// SIMATIC S7-200 project (STEP 7-Micro/WIN), CPU 222 REL 02.01

SYMBOL_TABLE USER1
E0               M0.0     // ESTADO 0
E1               M0.1     // ESTADO 1
E2               M0.2     // ESTADO 2
E3               M0.3     // ESTADO 3
E4               M0.4     // ESTADO 4
E5               M0.5     // ESTADO 5
E6               M0.6     // ESTADO 6
E7               M0.7     // ESTADO 7
E8               M1.0     // ESTADO 8
E9               M1.1     // ESTADO 9
E10              M1.2     // ESTADO 10
Esteira1         Q0.0     // Esteira 1
Esteira2         Q0.1     // Esteira2
S1               I0.0     // Sensor presença caixa pequena
S2               I0.1     // Sensor presença fim percurso
S3               I0.2     // Sensor presença caixa grande
S4               I0.3     // Sensor presença fim percuso
Cx1              Q0.2     // Gera caixa pequena
Cx2              Q0.3     // Gera caixa grande
Count1           VW200    // Quantidade caixas pequenas
Count2           VW210    // Quantidade caixas grandes
F1               M15.0    // Botão IHM
F2               M15.1    // Botão IHM
F3               M15.2    // Botão IHM
F4               M15.3    // Botao IHM
END_SYMBOL_TABLE
